// TIA Portal project "Projekt1" (V20)

(* hardware
DEVICE "GSD-Geraet_1"  GSD.Device.PN
   slot 0: "Baugruppenträger"  Rack  V1.0
   slot 0: "KRC4"  KRC4-ProfiNet_4.1  0x300  V4.1
      slot 0: "KRC4-ProfiNet_4.1"  KRC4-ProfiNet_4.1
      slot 1: "Interface1"  Interface1
         slot 1: "Port1"  Port1
   slot 1: "64 sichere digitale Ein- und Ausgänge_1"  64 safe digital in- and outputs  KUKA Device FIO64
      slot 0: "64 sichere digitale Ein- und Ausgänge"  64 safe digital in- and outputs
   slot 2: "256 digitale Ein- und Ausgänge_1"  256 digital in- and outputs  KUKA Device IO256
      slot 0: "256 digitale Ein- und Ausgänge"  256 digital in- and outputs
DEVICE "S7-1500/ET200MP-Station_1"  S7-1500 station
   slot 0: "Profilschiene_0"  Rack  6ES7 590-1***0-0AA0
   slot 1: "PLC_1"  CPU 1517F-3 PN  6ES7 517-3FQ10-0AB0  V4.0
      slot 3: "CPU-Display_1"  6ES7591-1BA00-0AA0
      slot 32768: "PROFINET-Schnittstelle_1"  X1
         slot 32769: "Port_1"  X1 P1
         slot 32770: "Port_2"  X1 P2
      slot 33024: "PROFINET-Schnittstelle_2"  X2
         slot 33025: "Port_1"  X2 P1
         slot 33026: "Port_2"  X2 P2
      slot 33280: "PROFINET-Schnittstelle GBIT_3"  X3
         slot 33281: "Port_1"  X3 P1
      slot 34817: "Virtual CP interface port_1"  Virtual CP interface port  Virtual CP interface port FW V4.0
DEVICE "GSD-Geraet_2"  GSD.Device.PN
   slot 0: "Baugruppenträger"  Rack  V1.0
   slot 0: "PN-PN-Coupler"  PN/PN Coupler X2  6ES7 158-3AD01-0XA0  V3.0
      slot 0: "PN/PN Coupler X2"  PN/PN Coupler X2
      slot 1: "PN-IO-02"  PN-IO-02
         slot 1: "Port 1"  Port 1
         slot 2: "Port 2"  Port 2
   slot 1: "PROFIsafe IN/OUT 12 Byte / 6 Byte_1"  PROFIsafe IN/OUT 12 Byte / 6 Byte
      slot 0: "PROFIsafe IN/OUT 12 Byte / 6 Byte"  PROFIsafe IN/OUT 12 Byte / 6 Byte
   slot 2: "PROFIsafe IN/OUT 6 Byte / 12 Byte_1"  PROFIsafe IN/OUT 6 Byte / 12 Byte
      slot 0: "PROFIsafe IN/OUT 6 Byte / 12 Byte"  PROFIsafe IN/OUT 6 Byte / 12 Byte
DEVICE "GSD-Geraet_3"  GSD.Device.PN
   slot 0: "Baugruppenträger"  Rack  V1.0
   slot 0: "PN-PN-Coupler_1"  PN/PN Coupler X1  6ES7 158-3AD01-0XA0  V3.0
      slot 0: "PN/PN Coupler X1"  PN/PN Coupler X1
      slot 1: "PN-IO-01"  PN-IO-01
         slot 1: "Port 1"  Port 1
         slot 2: "Port 2"  Port 2
   slot 1: "PROFIsafe IN/OUT 12 Byte / 6 Byte_1"  PROFIsafe IN/OUT 12 Byte / 6 Byte
      slot 0: "PROFIsafe IN/OUT 12 Byte / 6 Byte"  PROFIsafe IN/OUT 12 Byte / 6 Byte
   slot 2: "PROFIsafe IN/OUT 6 Byte / 12 Byte_1"  PROFIsafe IN/OUT 6 Byte / 12 Byte
      slot 0: "PROFIsafe IN/OUT 6 Byte / 12 Byte"  PROFIsafe IN/OUT 6 Byte / 12 Byte
*)

// ===== PLC "PLC_1"  CPU 1517F-3 PN =====

DATA_BLOCK "Main_Safety_RTG1_DB"   // DB1, F_DB
{ S7_Optimized_Access := 'TRUE' }
NAME : FUSI
VERSION : 0.1
// stored: InstanceOfName Main_Safety_RTG1
"Main_Safety_RTG1"
BEGIN
END_DATA_BLOCK

DATA_BLOCK "PositioningAxis_1"   // DB2, Motion_DB
{ S7_Optimized_Access := 'TRUE' }
AUTHOR : SIMATIC
FAMILY : MC_1500
VERSION : 9.0
// stored: InstanceOfName TO_PositioningAxis
"TO_PositioningAxis"
BEGIN
END_DATA_BLOCK

FUNCTION_BLOCK "Main_Safety_RTG1"   // FB1, F_FBD
{ S7_Optimized_Access := 'TRUE' }
BEGIN
END_FUNCTION_BLOCK

ORGANIZATION_BLOCK "Main"   // OB1, LAD, ProgramCycle
TITLE = "Main Program Sweep (Cycle)"
{ S7_Optimized_Access := 'TRUE' }
VERSION : 0.1
   VAR_INPUT
      Initial_Call : Bool;   // Initial call of this OB
      Remanence : Bool;   // =True, if remanent data are available
   END_VAR
BEGIN
END_ORGANIZATION_BLOCK